(* CoDeSys 2.3.9.31 project: 20161227.pro *)
(* Libraries: TcBase.lib 14.5.09 11:14:08, TcSystem.lib 27.2.12 14:08:36, TcBaseMath.lib 27.7.04 11:07:56, TcMath.lib 23.9.04 14:15:30, TcMC2.lib 23.8.12 10:01:14, STANDARD.LIB 5.6.98 11:03:02 *)

(* Task configuration *)
TASK Standard (PRIORITY := 0, INTERVAL := T#10ms);
	MAIN
END_TASK

(* Global variable list: Global_Variables *)
VAR_GLOBAL
	Axis1	:	Axis_Ref	;

END_VAR

(* Global variable list: TwinCAT_Configuration *)
(* Generated automatically by TwinCAT - (read only) *)
VAR_CONFIG
	MAIN.HomeInput1 AT %IX128.0 : BOOL;	(*  ~ {LinkedWith:TIID^Device 2 (EtherCAT)^Term 1 (EK1100)^Term 2 (EL1889)^Channel 1^Input} *)
	.Axis1.PlcToNc AT %QB0 : PLCTONC_AXIS_REF;	(*  ~ {LinkedWith:TINC^NC-Task 1 SAF^Axes^Axis 1^Inputs^Axis 1_FromPlc} *)
	.Axis1.NcToPlc AT %IB0 : NCTOPLC_AXIS_REF;	(*  ~ {LinkedWith:TINC^NC-Task 1 SAF^Axes^Axis 1^Outputs^Axis 1_ToPlc} *)
END_VAR

(* POU MAIN, ST *)
PROGRAM MAIN
VAR
	Enable : BOOL := TRUE;
	P1 : MC_Power;
	Move1: MC_MoveAbsolute;
	Home1:MC_Home;
	Home_Start : BOOL;
	HomeInput1 AT  %I*	:	BOOL;
	Home_Finish : BOOL;


	FuncNum: INT := -1;
	_FuncNum : INT := -1;
	Move_Finish : BOOL;
	Move_Start : BOOL := FALSE;
	t_1 :TON;
	start_t1_flag : BOOL := FALSE;
END_VAR
VAR PERSISTENT
	Position_x : ARRAY[1..9] OF REAL;
END_VAR
	P1(
	Enable:=Enable ,
	Enable_Positive:= TRUE,
	Enable_Negative:= TRUE ,
	Override:=100 ,
	Axis:= Axis1);

	Home1(
	Execute:= Home_Start,
	Position:= 0,
	bCalibrationCam:=HomeInput1 ,
	Axis:= Axis1,
	Done=>Home_Finish);


	Move1(
	Execute:=  Move_Start,
	Position:=Position_x[FuncNum],
	Velocity:=100 ,
	Axis:=Axis1 ,
	Done=>Move_Finish );

	IF start_t1_flag THEN
		t_1(IN:=start_t1_flag , PT:=t#0.1S  );
		IF t_1.Q THEN
			start_t1_flag := FALSE;
			Move_Start := TRUE;
		END_IF
	END_IF

	IF _FuncNum <> FuncNum THEN


		_FuncNum := FuncNum;
		CASE FuncNum OF
		1,2,3,4,5,6,7,8, 9 :
			Move_Start := FALSE;
			start_t1_flag := TRUE;



		ELSE

			FuncNum := -1;
			_FuncNum := -1;
		END_CASE;

	END_IF
END_PROGRAM
